{attribute 'GeneratedUsingTerminal: EL2502-0000-0016'}
{attribute addProperty BoxType "EL2502-0000-0016"}
{attribute addProperty Id "PWM_Outputs_Channel_1AT %Q*PWM_Outputs_Channel_4C6289CD2PWM_Outputs_Channel_2AT %Q*PWM_Outputs_Channel_4C6289CD2WcStateAT %I*WcState_0B2B16F91InfoDataAT %I*InfoData_94A18F5E2"}
{attribute addProperty CRC "2304954225"}
{attribute addProperty Size "7"}
TYPE EL2502_8962CF71 EXTENDS EtcSlaveTerminalBase_947E5A46 :
STRUCT
	{attribute addProperty Name "PWM_Outputs_Channel_1"}
	PWM_Outputs_Channel_1 : PWM_Outputs_Channel_4C6289CD;
	{attribute addProperty Name "PWM_Outputs_Channel_2"}
	PWM_Outputs_Channel_2 : PWM_Outputs_Channel_4C6289CD;
	{attribute addProperty Name "WcState"}
	WcState : WcState_0B2B16F9;
	{attribute addProperty Name "InfoData"}
	InfoData : InfoData_94A18F5E;
END_STRUCT
END_TYPE

(* stored: Version 1.2.0.0, ProductVersion 3.1.4024.9
   DUT EL2502_8962CF71: Id {2e2a10c6-42c7-4718-90fb-3360965ddeb8} *)
